{attribute 'GeneratedUsingTerminal: IODEVICETYPE_ETHERCATPROT'}
{attribute addProperty BoxType "IODEVICETYPE_ETHERCATPROT"}
{attribute addProperty Id "Beckhoff_EM2xxxBeckhoff_EM2xxx_23EB33C640Beckhoff_EM3xxxBeckhoff_EM3xxx_84530AF154Beckhoff_EM7xxxBeckhoff_EM7xxx_19818DAA633SyncUnitsSyncUnits_99E584AF18InputsInputs_25A0042B160OutputsOutputs_2397A10E106InfoDataInfoData_C76BEFB322"}
{attribute addProperty CRC "1966963591"}
{attribute addProperty Size "1033"}
TYPE EtherCAT_Master_EMxxxx_753D7B87 :
STRUCT
	{attribute addProperty Name "Beckhoff_EM2xxx"}
	{attribute addProperty PreviousPort "EtherCAT_Master_EMxxxx : Master"}
	Beckhoff_EM2xxx : Beckhoff_EM2xxx_23EB33C6;
	{attribute addProperty Name "Beckhoff_EM3xxx"}
	{attribute addProperty PreviousPort "Beckhoff EM2xxx : C"}
	Beckhoff_EM3xxx : Beckhoff_EM3xxx_84530AF1;
	{attribute addProperty Name "Beckhoff_EM7xxx"}
	{attribute addProperty PreviousPort "Beckhoff EM3xxx : C"}
	Beckhoff_EM7xxx : Beckhoff_EM7xxx_19818DAA;
	{attribute addProperty Name "SyncUnits"}
	SyncUnits : SyncUnits_99E584AF;
	{attribute addProperty Name "Inputs"}
	Inputs : Inputs_25A0042B;
	{attribute addProperty Name "Outputs"}
	Outputs : Outputs_2397A10E;
	{attribute addProperty Name "InfoData"}
	InfoData : InfoData_C76BEFB3;
END_STRUCT
END_TYPE

(* stored: Version 1.2.0.0, ProductVersion 3.1.4024.9
   DUT EtherCAT_Master_EMxxxx_753D7B87: Id {46050cb0-a94a-4e42-90ed-9bcf0c22b3c4} *)
